TYPE XtsHardwareStatus :
STRUCT
	AllMoversValid : BOOL;
	IsInSim : BOOL;
	ActiveMoverCount : UDINT;
	AreAllModulesInOp : BOOL;
	IsDCLinkVoltageReady : BOOL;
	AreAnyPartsInError : BOOL;
END_STRUCT
END_TYPE

(* stored: Version 1.1.0.1
   DUT XtsHardwareStatus: Id {94d3bf57-c2e0-40a2-beee-79ed0cbfb04f} *)
